(* IEC 61131-3 sources: SCADA-ICS-Security-101/Lab-02-ICS-SCADA-Architecture-Basics, 1 file *)

(* ---- plc_program.st ---- *)
PROGRAM PLC_PRG
VAR
    LED : BOOL;
END_VAR

LED := NOT LED;

END_PROGRAM
